(* Logix 5000 project; controller VET 1756-L62 rev 19.52; software revision 19.01; part 20 of 27 *)
(* tags used below, declared in another part *)
   estado : DINT[10];
   Batch : batch[10];
   comandos : DINT[10];
   dosificador : dosif_struct[20];
   Dosificar_LIQ_01 : PHASE;
   Dosificar_MAC_01 : PHASE;
   Dosificar_MAN_01 : PHASE;
   Dosificar_MIC_01 : PHASE;
(* Gestion_Dosificacion, continued *)

ROUTINE Reset_Local   (* ladder *)
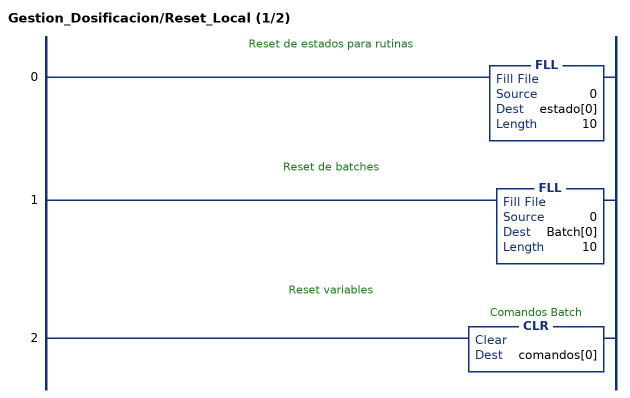
   // Reset de estados para rutinas
   0: FLL(0,estado[0],10);
   // Reset de batches
   1: FLL(0,Batch[0],10);
   // Reset variables
   2: CLR(comandos[0]);
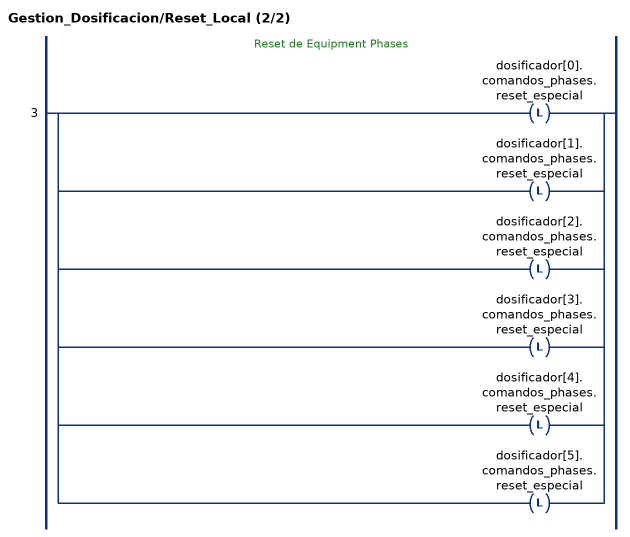
   // Reset de Equipment Phases
   3: [OTL(dosificador[0].comandos_phases.reset_especial) ,OTL(dosificador[1].comandos_phases.reset_especial) ,OTL(dosificador[2].comandos_phases.reset_especial) ,OTL(dosificador[3].comandos_phases.reset_especial) ,OTL(dosificador[4].comandos_phases.reset_especial) ,OTL(dosificador[5].comandos_phases.reset_especial) ];
END_ROUTINE
END_PROGRAM

PROGRAM Interfaz_Equipment_Phase   (* main routine main *)

ROUTINE Dosificar_LIQ_01   (* ladder *)
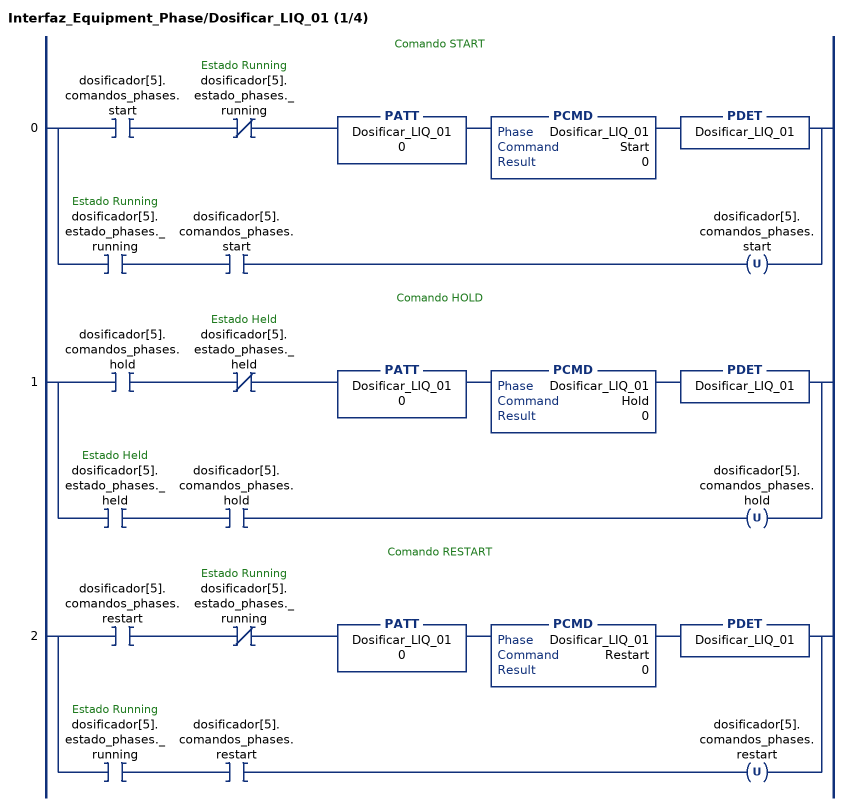
   // Comando START
   0: [XIC(dosificador[5].comandos_phases.start) XIO(dosificador[5].estado_phases._running) PATT(Dosificar_LIQ_01,0) PCMD(Dosificar_LIQ_01,Start,0) PDET(Dosificar_LIQ_01) ,XIC(dosificador[5].estado_phases._running) XIC(dosificador[5].comandos_phases.start) OTU(dosificador[5].comandos_phases.start) ];
   // Comando HOLD
   1: [XIC(dosificador[5].comandos_phases.hold) XIO(dosificador[5].estado_phases._held) PATT(Dosificar_LIQ_01,0) PCMD(Dosificar_LIQ_01,Hold,0) PDET(Dosificar_LIQ_01) ,XIC(dosificador[5].estado_phases._held) XIC(dosificador[5].comandos_phases.hold) OTU(dosificador[5].comandos_phases.hold) ];
   // Comando RESTART
   2: [XIC(dosificador[5].comandos_phases.restart) XIO(dosificador[5].estado_phases._running) PATT(Dosificar_LIQ_01,0) PCMD(Dosificar_LIQ_01,Restart,0) PDET(Dosificar_LIQ_01) ,XIC(dosificador[5].estado_phases._running) XIC(dosificador[5].comandos_phases.restart) OTU(dosificador[5].comandos_phases.restart) ];
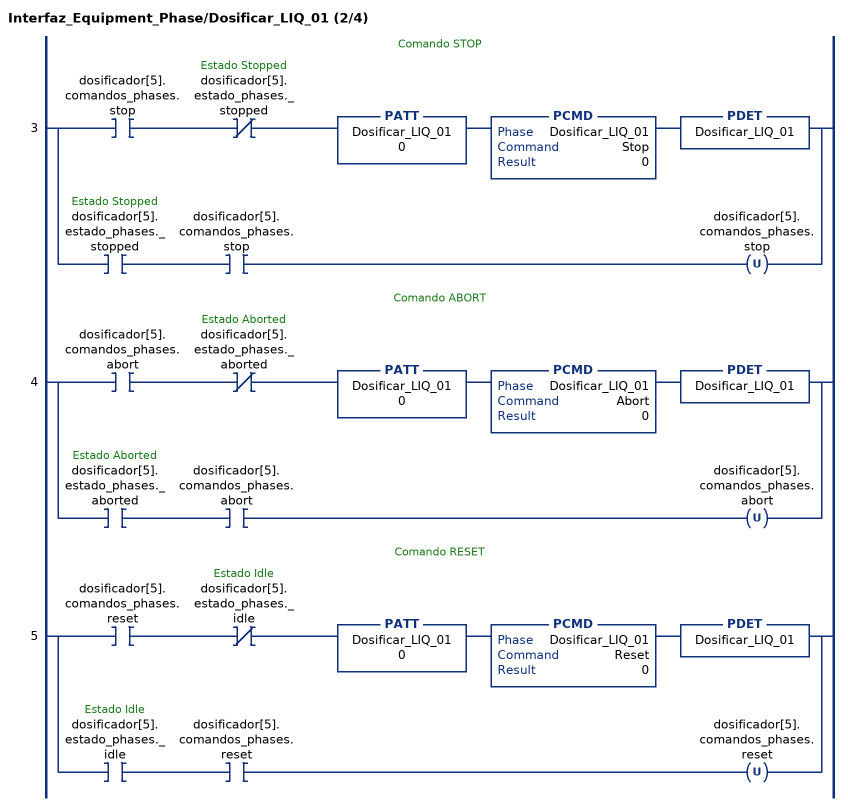
   // Comando STOP
   3: [XIC(dosificador[5].comandos_phases.stop) XIO(dosificador[5].estado_phases._stopped) PATT(Dosificar_LIQ_01,0) PCMD(Dosificar_LIQ_01,Stop,0) PDET(Dosificar_LIQ_01) ,XIC(dosificador[5].estado_phases._stopped) XIC(dosificador[5].comandos_phases.stop) OTU(dosificador[5].comandos_phases.stop) ];
   // Comando ABORT
   4: [XIC(dosificador[5].comandos_phases.abort) XIO(dosificador[5].estado_phases._aborted) PATT(Dosificar_LIQ_01,0) PCMD(Dosificar_LIQ_01,Abort,0) PDET(Dosificar_LIQ_01) ,XIC(dosificador[5].estado_phases._aborted) XIC(dosificador[5].comandos_phases.abort) OTU(dosificador[5].comandos_phases.abort) ];
   // Comando RESET
   5: [XIC(dosificador[5].comandos_phases.reset) XIO(dosificador[5].estado_phases._idle) PATT(Dosificar_LIQ_01,0) PCMD(Dosificar_LIQ_01,Reset,0) PDET(Dosificar_LIQ_01) ,XIC(dosificador[5].estado_phases._idle) XIC(dosificador[5].comandos_phases.reset) OTU(dosificador[5].comandos_phases.reset) ];
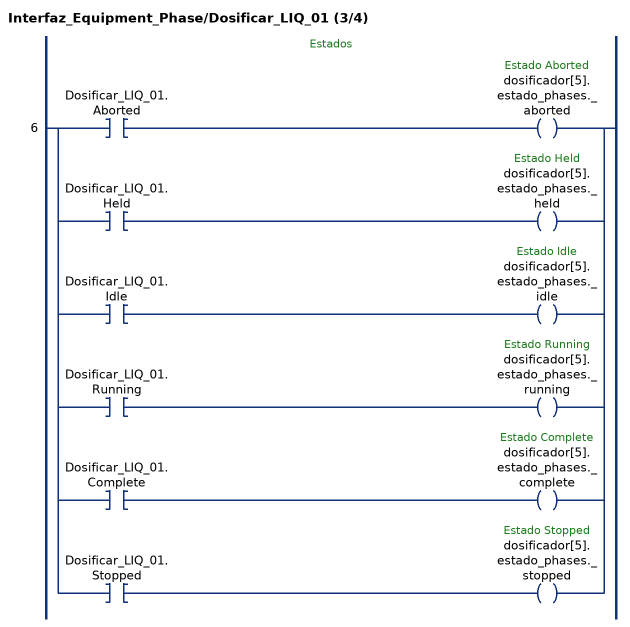
   // Estados
   6: [XIC(Dosificar_LIQ_01.Aborted) OTE(dosificador[5].estado_phases._aborted) ,XIC(Dosificar_LIQ_01.Held) OTE(dosificador[5].estado_phases._held) ,XIC(Dosificar_LIQ_01.Idle) OTE(dosificador[5].estado_phases._idle) ,XIC(Dosificar_LIQ_01.Running) OTE(dosificador[5].estado_phases._running) ,XIC(Dosificar_LIQ_01.Complete) OTE(dosificador[5].estado_phases._complete) ,XIC(Dosificar_LIQ_01.Stopped) OTE(dosificador[5].estado_phases._stopped) ];
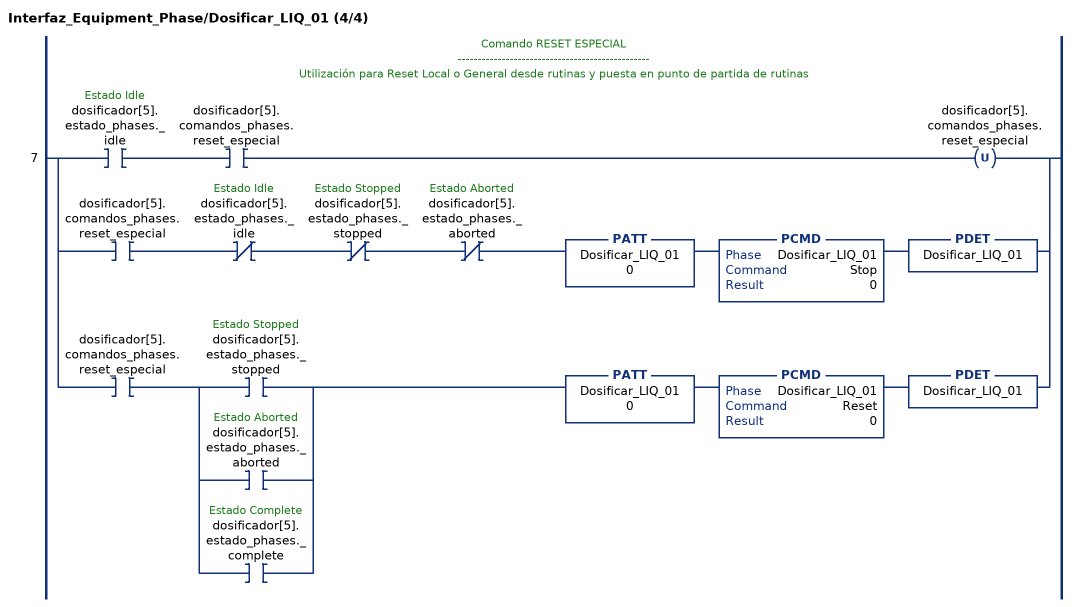
   // Comando RESET ESPECIAL
   // ------------------------------------------------
   // Utilización para Reset Local o General desde rutinas y puesta en punto de partida de rutinas
   7: [XIC(dosificador[5].estado_phases._idle) XIC(dosificador[5].comandos_phases.reset_especial) OTU(dosificador[5].comandos_phases.reset_especial) ,XIC(dosificador[5].comandos_phases.reset_especial) XIO(dosificador[5].estado_phases._idle) XIO(dosificador[5].estado_phases._stopped) XIO(dosificador[5].estado_phases._aborted) PATT(Dosificar_LIQ_01,0) PCMD(Dosificar_LIQ_01,Stop,0) PDET(Dosificar_LIQ_01) ,XIC(dosificador[5].comandos_phases.reset_especial) [XIC(dosificador[5].estado_phases._stopped) ,XIC(dosificador[5].estado_phases._aborted) ,XIC(dosificador[5].estado_phases._complete) ] PATT(Dosificar_LIQ_01,0) PCMD(Dosificar_LIQ_01,Reset,0) PDET(Dosificar_LIQ_01) ];
END_ROUTINE

ROUTINE Dosificar_MAC_01   (* ladder *)
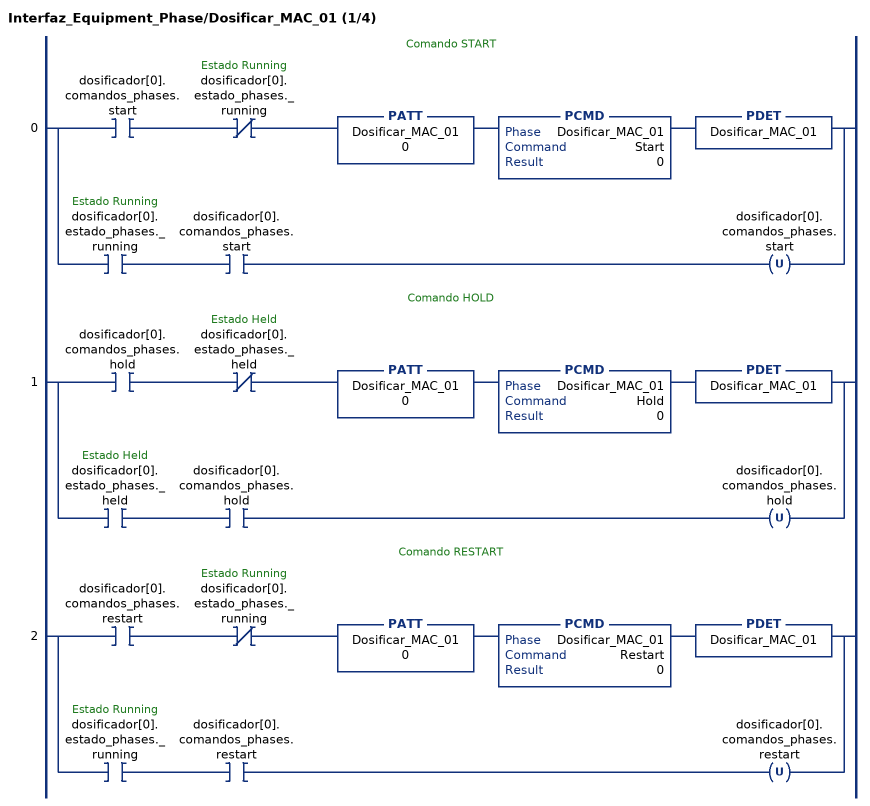
   // Comando START
   0: [XIC(dosificador[0].comandos_phases.start) XIO(dosificador[0].estado_phases._running) PATT(Dosificar_MAC_01,0) PCMD(Dosificar_MAC_01,Start,0) PDET(Dosificar_MAC_01) ,XIC(dosificador[0].estado_phases._running) XIC(dosificador[0].comandos_phases.start) OTU(dosificador[0].comandos_phases.start) ];
   // Comando HOLD
   1: [XIC(dosificador[0].comandos_phases.hold) XIO(dosificador[0].estado_phases._held) PATT(Dosificar_MAC_01,0) PCMD(Dosificar_MAC_01,Hold,0) PDET(Dosificar_MAC_01) ,XIC(dosificador[0].estado_phases._held) XIC(dosificador[0].comandos_phases.hold) OTU(dosificador[0].comandos_phases.hold) ];
   // Comando RESTART
   2: [XIC(dosificador[0].comandos_phases.restart) XIO(dosificador[0].estado_phases._running) PATT(Dosificar_MAC_01,0) PCMD(Dosificar_MAC_01,Restart,0) PDET(Dosificar_MAC_01) ,XIC(dosificador[0].estado_phases._running) XIC(dosificador[0].comandos_phases.restart) OTU(dosificador[0].comandos_phases.restart) ];
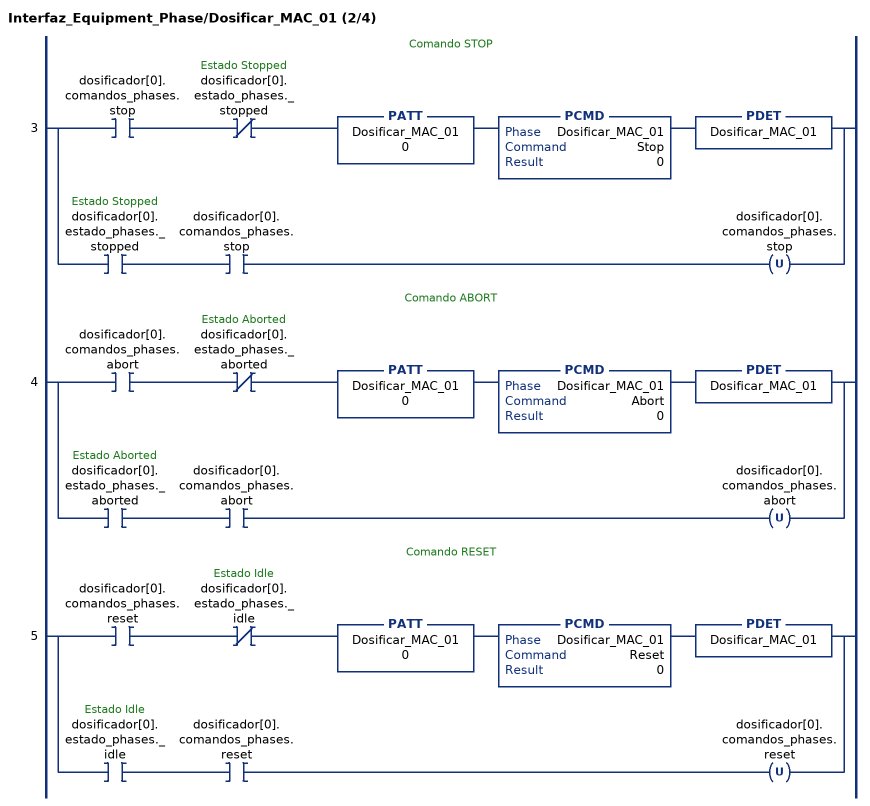
   // Comando STOP
   3: [XIC(dosificador[0].comandos_phases.stop) XIO(dosificador[0].estado_phases._stopped) PATT(Dosificar_MAC_01,0) PCMD(Dosificar_MAC_01,Stop,0) PDET(Dosificar_MAC_01) ,XIC(dosificador[0].estado_phases._stopped) XIC(dosificador[0].comandos_phases.stop) OTU(dosificador[0].comandos_phases.stop) ];
   // Comando ABORT
   4: [XIC(dosificador[0].comandos_phases.abort) XIO(dosificador[0].estado_phases._aborted) PATT(Dosificar_MAC_01,0) PCMD(Dosificar_MAC_01,Abort,0) PDET(Dosificar_MAC_01) ,XIC(dosificador[0].estado_phases._aborted) XIC(dosificador[0].comandos_phases.abort) OTU(dosificador[0].comandos_phases.abort) ];
   // Comando RESET
   5: [XIC(dosificador[0].comandos_phases.reset) XIO(dosificador[0].estado_phases._idle) PATT(Dosificar_MAC_01,0) PCMD(Dosificar_MAC_01,Reset,0) PDET(Dosificar_MAC_01) ,XIC(dosificador[0].estado_phases._idle) XIC(dosificador[0].comandos_phases.reset) OTU(dosificador[0].comandos_phases.reset) ];
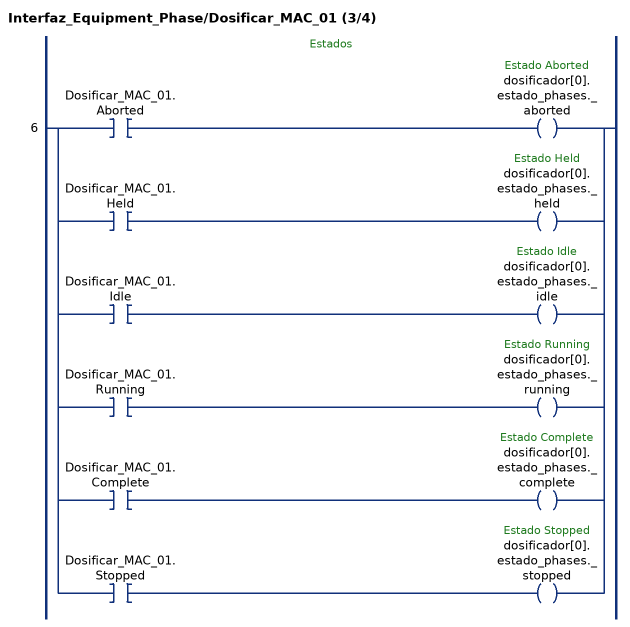
   // Estados
   6: [XIC(Dosificar_MAC_01.Aborted) OTE(dosificador[0].estado_phases._aborted) ,XIC(Dosificar_MAC_01.Held) OTE(dosificador[0].estado_phases._held) ,XIC(Dosificar_MAC_01.Idle) OTE(dosificador[0].estado_phases._idle) ,XIC(Dosificar_MAC_01.Running) OTE(dosificador[0].estado_phases._running) ,XIC(Dosificar_MAC_01.Complete) OTE(dosificador[0].estado_phases._complete) ,XIC(Dosificar_MAC_01.Stopped) OTE(dosificador[0].estado_phases._stopped) ];
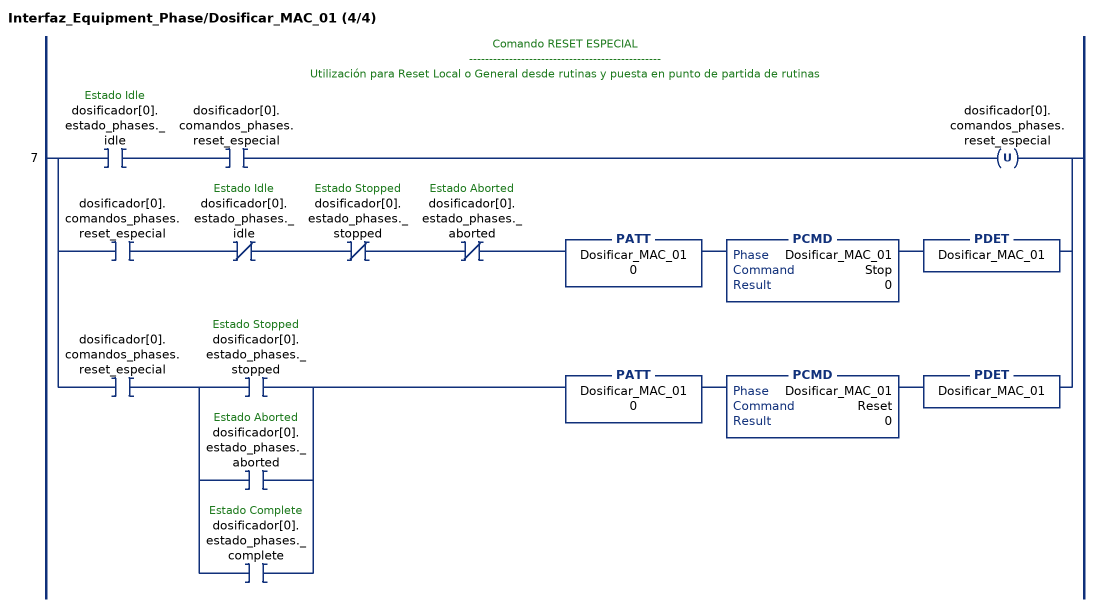
   // Comando RESET ESPECIAL
   // ------------------------------------------------
   // Utilización para Reset Local o General desde rutinas y puesta en punto de partida de rutinas
   7: [XIC(dosificador[0].estado_phases._idle) XIC(dosificador[0].comandos_phases.reset_especial) OTU(dosificador[0].comandos_phases.reset_especial) ,XIC(dosificador[0].comandos_phases.reset_especial) XIO(dosificador[0].estado_phases._idle) XIO(dosificador[0].estado_phases._stopped) XIO(dosificador[0].estado_phases._aborted) PATT(Dosificar_MAC_01,0) PCMD(Dosificar_MAC_01,Stop,0) PDET(Dosificar_MAC_01) ,XIC(dosificador[0].comandos_phases.reset_especial) [XIC(dosificador[0].estado_phases._stopped) ,XIC(dosificador[0].estado_phases._aborted) ,XIC(dosificador[0].estado_phases._complete) ] PATT(Dosificar_MAC_01,0) PCMD(Dosificar_MAC_01,Reset,0) PDET(Dosificar_MAC_01) ];
END_ROUTINE

ROUTINE Dosificar_MAN_01   (* ladder *)
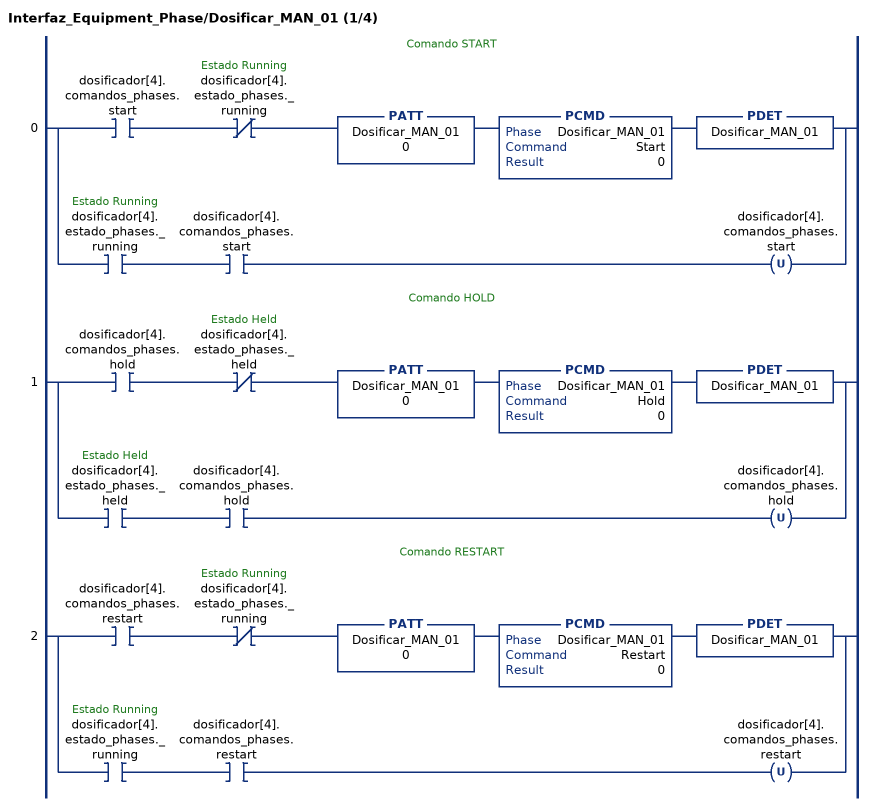
   // Comando START
   0: [XIC(dosificador[4].comandos_phases.start) XIO(dosificador[4].estado_phases._running) PATT(Dosificar_MAN_01,0) PCMD(Dosificar_MAN_01,Start,0) PDET(Dosificar_MAN_01) ,XIC(dosificador[4].estado_phases._running) XIC(dosificador[4].comandos_phases.start) OTU(dosificador[4].comandos_phases.start) ];
   // Comando HOLD
   1: [XIC(dosificador[4].comandos_phases.hold) XIO(dosificador[4].estado_phases._held) PATT(Dosificar_MAN_01,0) PCMD(Dosificar_MAN_01,Hold,0) PDET(Dosificar_MAN_01) ,XIC(dosificador[4].estado_phases._held) XIC(dosificador[4].comandos_phases.hold) OTU(dosificador[4].comandos_phases.hold) ];
   // Comando RESTART
   2: [XIC(dosificador[4].comandos_phases.restart) XIO(dosificador[4].estado_phases._running) PATT(Dosificar_MAN_01,0) PCMD(Dosificar_MAN_01,Restart,0) PDET(Dosificar_MAN_01) ,XIC(dosificador[4].estado_phases._running) XIC(dosificador[4].comandos_phases.restart) OTU(dosificador[4].comandos_phases.restart) ];
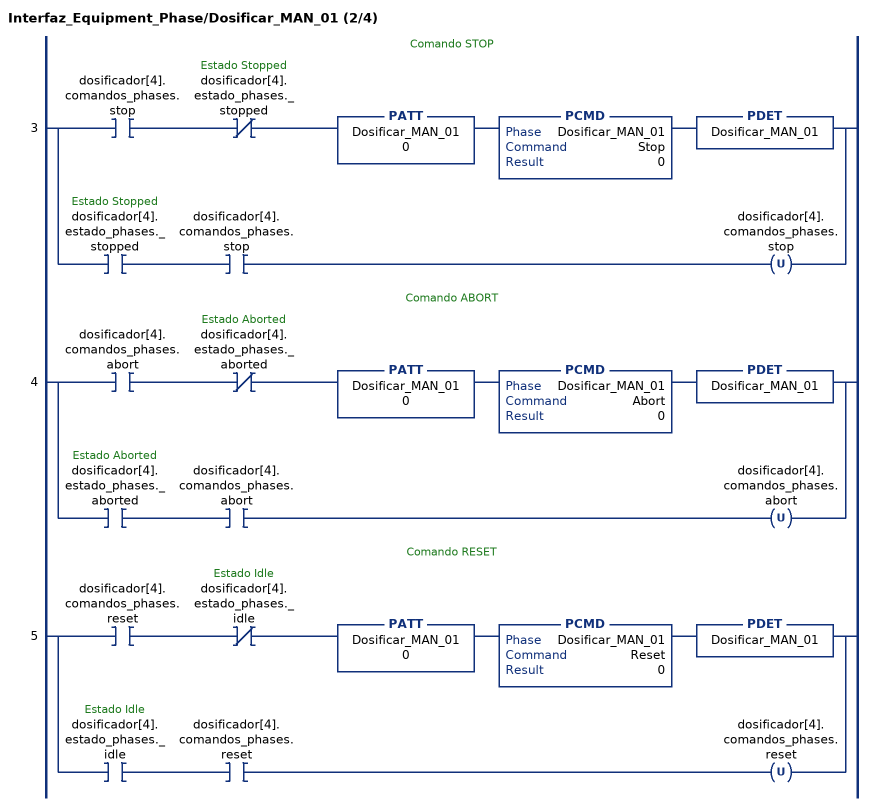
   // Comando STOP
   3: [XIC(dosificador[4].comandos_phases.stop) XIO(dosificador[4].estado_phases._stopped) PATT(Dosificar_MAN_01,0) PCMD(Dosificar_MAN_01,Stop,0) PDET(Dosificar_MAN_01) ,XIC(dosificador[4].estado_phases._stopped) XIC(dosificador[4].comandos_phases.stop) OTU(dosificador[4].comandos_phases.stop) ];
   // Comando ABORT
   4: [XIC(dosificador[4].comandos_phases.abort) XIO(dosificador[4].estado_phases._aborted) PATT(Dosificar_MAN_01,0) PCMD(Dosificar_MAN_01,Abort,0) PDET(Dosificar_MAN_01) ,XIC(dosificador[4].estado_phases._aborted) XIC(dosificador[4].comandos_phases.abort) OTU(dosificador[4].comandos_phases.abort) ];
   // Comando RESET
   5: [XIC(dosificador[4].comandos_phases.reset) XIO(dosificador[4].estado_phases._idle) PATT(Dosificar_MAN_01,0) PCMD(Dosificar_MAN_01,Reset,0) PDET(Dosificar_MAN_01) ,XIC(dosificador[4].estado_phases._idle) XIC(dosificador[4].comandos_phases.reset) OTU(dosificador[4].comandos_phases.reset) ];
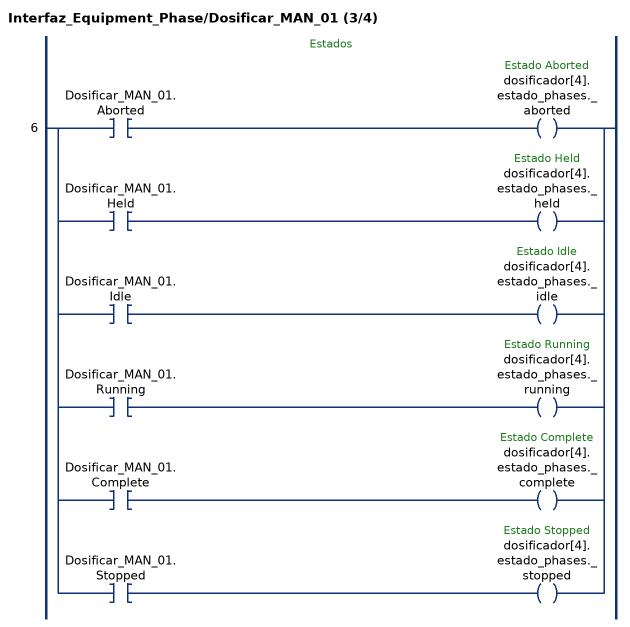
   // Estados
   6: [XIC(Dosificar_MAN_01.Aborted) OTE(dosificador[4].estado_phases._aborted) ,XIC(Dosificar_MAN_01.Held) OTE(dosificador[4].estado_phases._held) ,XIC(Dosificar_MAN_01.Idle) OTE(dosificador[4].estado_phases._idle) ,XIC(Dosificar_MAN_01.Running) OTE(dosificador[4].estado_phases._running) ,XIC(Dosificar_MAN_01.Complete) OTE(dosificador[4].estado_phases._complete) ,XIC(Dosificar_MAN_01.Stopped) OTE(dosificador[4].estado_phases._stopped) ];
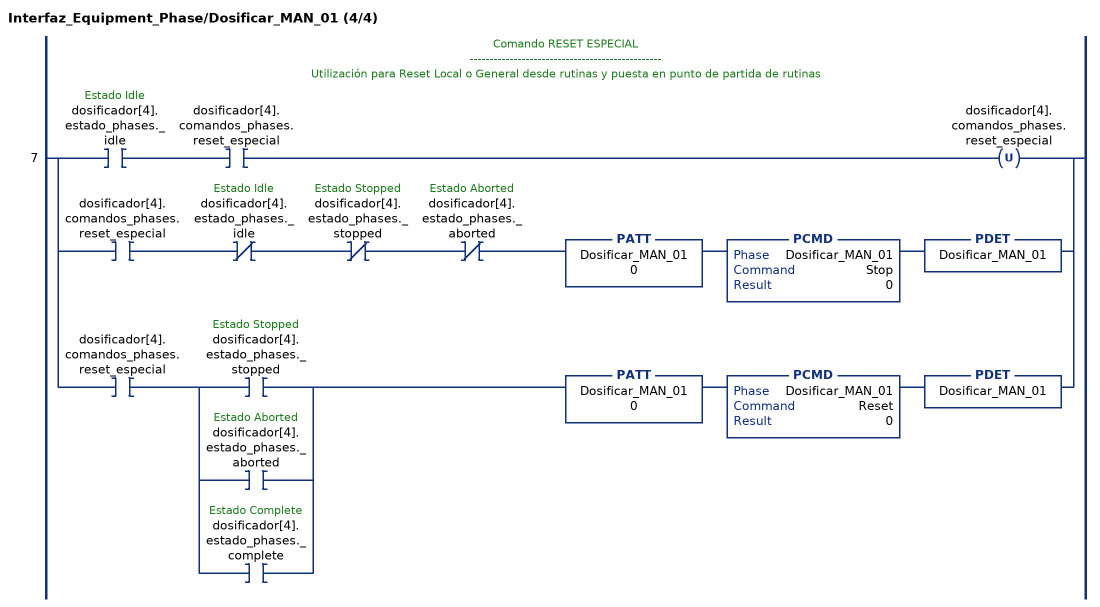
   // Comando RESET ESPECIAL
   // ------------------------------------------------
   // Utilización para Reset Local o General desde rutinas y puesta en punto de partida de rutinas
   7: [XIC(dosificador[4].estado_phases._idle) XIC(dosificador[4].comandos_phases.reset_especial) OTU(dosificador[4].comandos_phases.reset_especial) ,XIC(dosificador[4].comandos_phases.reset_especial) XIO(dosificador[4].estado_phases._idle) XIO(dosificador[4].estado_phases._stopped) XIO(dosificador[4].estado_phases._aborted) PATT(Dosificar_MAN_01,0) PCMD(Dosificar_MAN_01,Stop,0) PDET(Dosificar_MAN_01) ,XIC(dosificador[4].comandos_phases.reset_especial) [XIC(dosificador[4].estado_phases._stopped) ,XIC(dosificador[4].estado_phases._aborted) ,XIC(dosificador[4].estado_phases._complete) ] PATT(Dosificar_MAN_01,0) PCMD(Dosificar_MAN_01,Reset,0) PDET(Dosificar_MAN_01) ];
END_ROUTINE

ROUTINE Dosificar_MIC_01   (* ladder *)
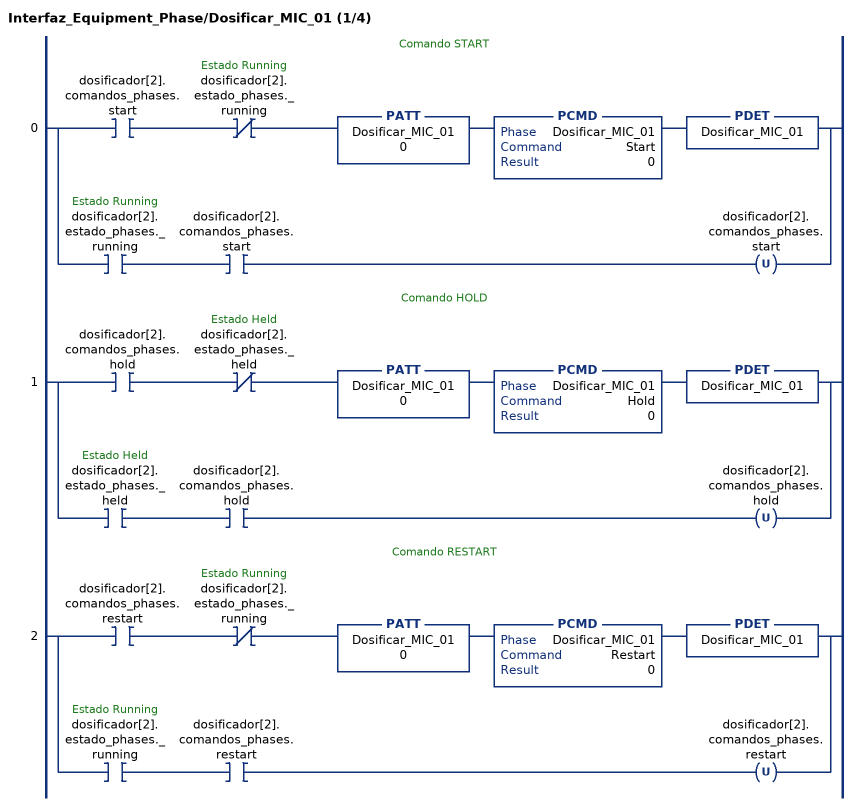
   // Comando START
   0: [XIC(dosificador[2].comandos_phases.start) XIO(dosificador[2].estado_phases._running) PATT(Dosificar_MIC_01,0) PCMD(Dosificar_MIC_01,Start,0) PDET(Dosificar_MIC_01) ,XIC(dosificador[2].estado_phases._running) XIC(dosificador[2].comandos_phases.start) OTU(dosificador[2].comandos_phases.start) ];
   // Comando HOLD
   1: [XIC(dosificador[2].comandos_phases.hold) XIO(dosificador[2].estado_phases._held) PATT(Dosificar_MIC_01,0) PCMD(Dosificar_MIC_01,Hold,0) PDET(Dosificar_MIC_01) ,XIC(dosificador[2].estado_phases._held) XIC(dosificador[2].comandos_phases.hold) OTU(dosificador[2].comandos_phases.hold) ];
   // Comando RESTART
   2: [XIC(dosificador[2].comandos_phases.restart) XIO(dosificador[2].estado_phases._running) PATT(Dosificar_MIC_01,0) PCMD(Dosificar_MIC_01,Restart,0) PDET(Dosificar_MIC_01) ,XIC(dosificador[2].estado_phases._running) XIC(dosificador[2].comandos_phases.restart) OTU(dosificador[2].comandos_phases.restart) ];
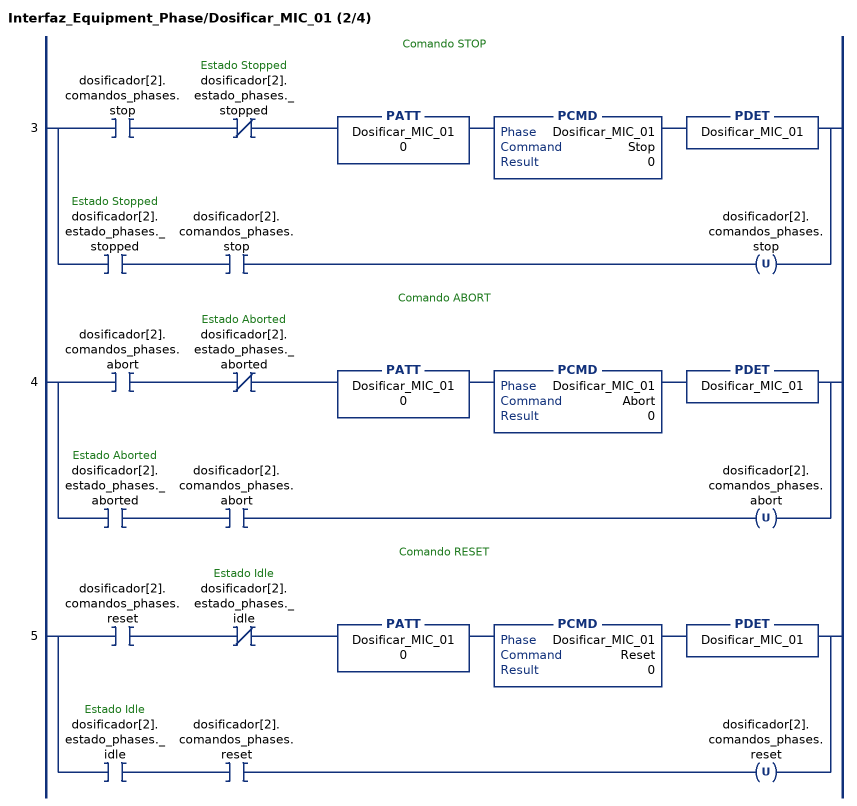
   // Comando STOP
   3: [XIC(dosificador[2].comandos_phases.stop) XIO(dosificador[2].estado_phases._stopped) PATT(Dosificar_MIC_01,0) PCMD(Dosificar_MIC_01,Stop,0) PDET(Dosificar_MIC_01) ,XIC(dosificador[2].estado_phases._stopped) XIC(dosificador[2].comandos_phases.stop) OTU(dosificador[2].comandos_phases.stop) ];
   // Comando ABORT
   4: [XIC(dosificador[2].comandos_phases.abort) XIO(dosificador[2].estado_phases._aborted) PATT(Dosificar_MIC_01,0) PCMD(Dosificar_MIC_01,Abort,0) PDET(Dosificar_MIC_01) ,XIC(dosificador[2].estado_phases._aborted) XIC(dosificador[2].comandos_phases.abort) OTU(dosificador[2].comandos_phases.abort) ];
   // Comando RESET
   5: [XIC(dosificador[2].comandos_phases.reset) XIO(dosificador[2].estado_phases._idle) PATT(Dosificar_MIC_01,0) PCMD(Dosificar_MIC_01,Reset,0) PDET(Dosificar_MIC_01) ,XIC(dosificador[2].estado_phases._idle) XIC(dosificador[2].comandos_phases.reset) OTU(dosificador[2].comandos_phases.reset) ];
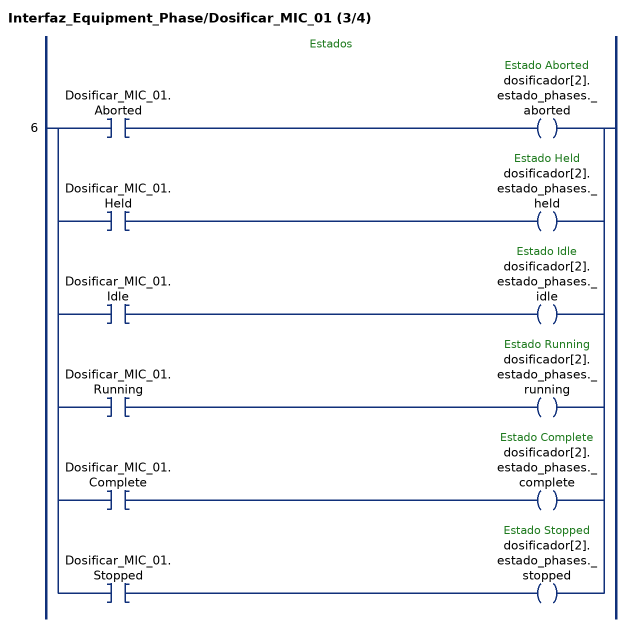
   // Estados
   6: [XIC(Dosificar_MIC_01.Aborted) OTE(dosificador[2].estado_phases._aborted) ,XIC(Dosificar_MIC_01.Held) OTE(dosificador[2].estado_phases._held) ,XIC(Dosificar_MIC_01.Idle) OTE(dosificador[2].estado_phases._idle) ,XIC(Dosificar_MIC_01.Running) OTE(dosificador[2].estado_phases._running) ,XIC(Dosificar_MIC_01.Complete) OTE(dosificador[2].estado_phases._complete) ,XIC(Dosificar_MIC_01.Stopped) OTE(dosificador[2].estado_phases._stopped) ];
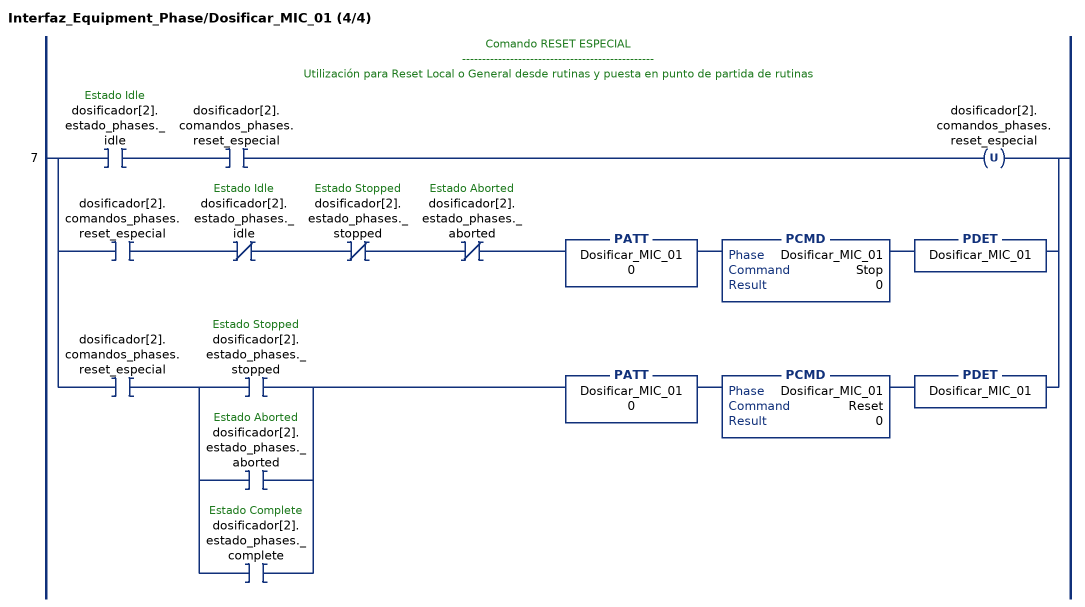
   // Comando RESET ESPECIAL
   // ------------------------------------------------
   // Utilización para Reset Local o General desde rutinas y puesta en punto de partida de rutinas
   7: [XIC(dosificador[2].estado_phases._idle) XIC(dosificador[2].comandos_phases.reset_especial) OTU(dosificador[2].comandos_phases.reset_especial) ,XIC(dosificador[2].comandos_phases.reset_especial) XIO(dosificador[2].estado_phases._idle) XIO(dosificador[2].estado_phases._stopped) XIO(dosificador[2].estado_phases._aborted) PATT(Dosificar_MIC_01,0) PCMD(Dosificar_MIC_01,Stop,0) PDET(Dosificar_MIC_01) ,XIC(dosificador[2].comandos_phases.reset_especial) [XIC(dosificador[2].estado_phases._stopped) ,XIC(dosificador[2].estado_phases._aborted) ,XIC(dosificador[2].estado_phases._complete) ] PATT(Dosificar_MIC_01,0) PCMD(Dosificar_MIC_01,Reset,0) PDET(Dosificar_MIC_01) ];
END_ROUTINE
